// TIA Portal V21 export
VAR_GLOBAL   // PLC tag table "SmokeTags"
   Smoke_Bit AT %M10.0 : Bool;
   Smoke_Out AT %M10.1 : Bool;
   Smoke_Int AT %MW12 : Int;
END_VAR
